// Block: A0302_Rulliera_PERS

DATA_BLOCK A0302_Rulliera_PERS
VERSION : 0.1
   NON_RETAIN
   VAR
      Par : Struct
         Ax : SpeedMachine_Par;
         Ax_Aut : A0301_Mach_Speed_Par;
      END_STRUCT;
      IEC_SP : Struct
         FTC_CodaRall : Struct
            TON_PT : Time;
            TOF_PT : Time;
         END_STRUCT;
         FTC_CodaProxIng : Struct
            TON_PT : Time;
            TOF_PT : Time;
         END_STRUCT;
         FTC_Centro : Struct
            TON_PT : Time;
            TOF_PT : Time;
         END_STRUCT;
      END_STRUCT;
   END_VAR

BEGIN
   // No initialization required
END_DATA_BLOCK
